(* IEC 61131-3 sources: ldsoft/build/bin, 1 file *)

(* ---- cc.st ---- *)
(* 梯形图生成的ST代码 *)
PROGRAM LadderProgram

VAR
    Start : BOOL;
    Stop : BOOL;
    Motor : BOOL;
END_VAR

(* 主程序 *)
Motor := Start AND NOT Stop;

END_PROGRAM
